// TIA Portal project "Project2" (V16)

(* hardware
DEVICE "S7300/ET200M station_1"  S7-300 station
   slot 0: "Rail_0"  Rail  6ES7 390-1***0-0AA0
   slot 2: "PLC_1"  CPU 313C-2 DP  6ES7 313-6CF03-0AB0  V2.6
      slot 0: "MPI interface_1"  X1
      slot 1: "DP interface_1"  X2
      slot 2: "DI 16/DO 16_1"  DI16/DO16
      slot 4: "Count_1"  Counter
*)

// ===== PLC "PLC_1"  CPU 313C-2 DP =====

VAR_GLOBAL   // PLC tag table "Default tag table"
   "Start - Moto1" AT %I0.0 : Bool;
   "Stop - Moto1" AT %I0.1 : Bool;
   "Oload1" AT %I0.2 : Bool;
   "Start - Moto2" AT %I0.3 : Bool;
   "Stop - Moto2" AT %I0.4 : Bool;
   "Oload2" AT %I0.5 : Bool;
   "Motor1" AT %Q0.0 : Bool;
   "Motor2" AT %Q0.1 : Bool;
   "Moto1 - led" AT %Q0.2 : Bool;
   "Moto2 - led" AT %Q0.3 : Bool;
END_VAR

ORGANIZATION_BLOCK "Main"   // OB1, LAD
TITLE = "Main Program Sweep (Cycle)"
{ S7_Optimized_Access := 'FALSE' }
VERSION : 0.1
   VAR_TEMP
      OB1_EV_CLASS : Byte;   // Bits 0-3 = 1 (Coming event), Bits 4-7 = 1 (Event class 1)
      OB1_SCAN_1 : Byte;   // 1 (Cold restart scan 1 of OB 1), 3 (Scan 2-n of OB 1)
      OB1_PRIORITY : Byte;   // Priority of OB Execution
      OB1_OB_NUMBR : Byte;   // 1 (Organization block 1, OB1)
      OB1_RESERVED_1 : Byte;   // Reserved for system
      OB1_RESERVED_2 : Byte;   // Reserved for system
      OB1_PREV_CYCLE : Int;   // Cycle time of previous OB1 scan (milliseconds)
      OB1_MIN_CYCLE : Int;   // Minimum cycle time of OB1 (milliseconds)
      OB1_MAX_CYCLE : Int;   // Maximum cycle time of OB1 (milliseconds)
      OB1_DATE_TIME : Date_And_Time;   // Date and time OB1 started
   END_VAR
BEGIN

REGION Network 1: Motor 1
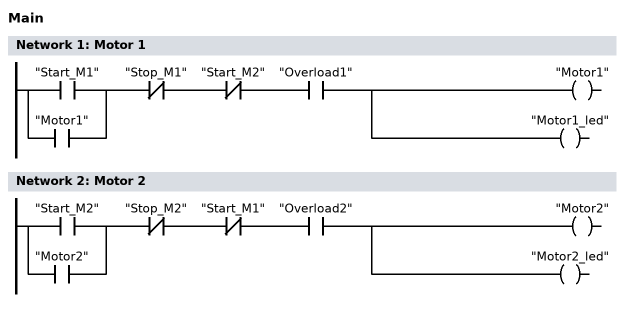
   RUNG wire#powerrail
      Contact( "Start_M1" )
      wire#w1
      I_Contact( "Stop_M1" )
      I_Contact( "Start_M2" )
      Contact( "Overload1" )
      wire#w2
      Coil( "Motor1" )
   END_RUNG
   RUNG wire#powerrail
      Contact( "Motor1" )
   END_RUNG wire#w1
   RUNG wire#w2
      Coil( "Motor1_led" )
   END_RUNG
   // the same network as SCL:
   "Motor1" := ("Start_M1" OR "Motor1") AND NOT "Stop_M1" AND NOT "Start_M2" AND "Overload1";
   "Motor1_led" := "Motor1";
END_REGION

REGION Network 2: Motor 2
   RUNG wire#powerrail
      Contact( "Start_M2" )
      wire#w1
      I_Contact( "Stop_M2" )
      I_Contact( "Start_M1" )
      Contact( "Overload2" )
      wire#w2
      Coil( "Motor2" )
   END_RUNG
   RUNG wire#powerrail
      Contact( "Motor2" )
   END_RUNG wire#w1
   RUNG wire#w2
      Coil( "Motor2_led" )
   END_RUNG
   // the same network as SCL:
   "Motor2" := ("Start_M2" OR "Motor2") AND NOT "Stop_M2" AND NOT "Start_M1" AND "Overload2";
   "Motor2_led" := "Motor2";
END_REGION
END_ORGANIZATION_BLOCK